# EPICS substitutions: db/ecat2el3602.substitutions
file ecat2slave.template
{
	pattern {DEVICENAME}
		{EL3602}
}

file ecat2el360xel320x.template
{
	pattern {CH_ID, PDO_IDX, ESLO}
		{$(MOD_ID)-AI1, 0, 0.000000004656612873077392578}
		{$(MOD_ID)-AI2, 1, 0.000000004656612873077392578}
}
